(* PLC project power_supply, Dassault Systèmes ControlBuild 2024x *)
(* stored: creationDateTime 2023-10-03T11:13:22-01:00 *)

(* This module simulates a transformation of electrical energy : power supply. *)
FUNCTION_BLOCK equipment_library.power_supply
  VAR_INPUT
    inputEnergy : BOOL := true;
  END_VAR
  VAR_OUTPUT
    outputEnergy : BOOL := false;
  END_VAR
  VAR
    d_electrical : BOOL := false;
    v_d_electrical : BOOL := false;
  END_VAR


ACTION C_source_code:
/* ----------------------------------------------------------------	*/
/* Type : Model of Operative Behaviour					*/
/* Category :  Power								*/
/* Author : Dassault Systemes						*/
/* Update date : June 2018							*/
/* ----------------------------------------------------------------	*/
/* This module simulates a transformation of electrical energy.  	*/
/* This simulates a power supply.						*/
/* ----------------------------------------------------------------	*/

if (d_electrical)
	outputEnergy = v_d_electrical;

else		/* 	else it returns the input value 			*/
	outputEnergy = inputEnergy;
END_ACTION
END_FUNCTION_BLOCK
